FUNCTION_BLOCK NeredaSludgeBuffer (* Composite Function Block Type *)
  (* Standard: 61499-2 *)
  (* Version 0.0, 4/25/2024, SESA713705, Schneider Electric, template *)
  PACKAGE SE.Nereda;
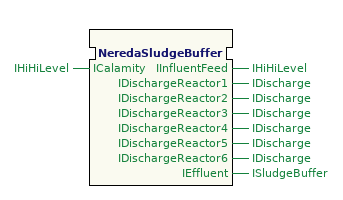
  SOCKETS
    ICalamity : IHiHiLevel;
  END_SOCKETS
  PLUGS
    IInfluentFeed : IHiHiLevel;
    IDischargeReactor1 : IDischarge;
    IDischargeReactor2 : IDischarge;
    IDischargeReactor3 : IDischarge;
    IDischargeReactor4 : IDischarge;
    IDischargeReactor5 : IDischarge;
    IDischargeReactor6 : IDischarge;
    IEffluent : ISludgeBuffer; (* Process value and status interface adapter *)
  END_PLUGS
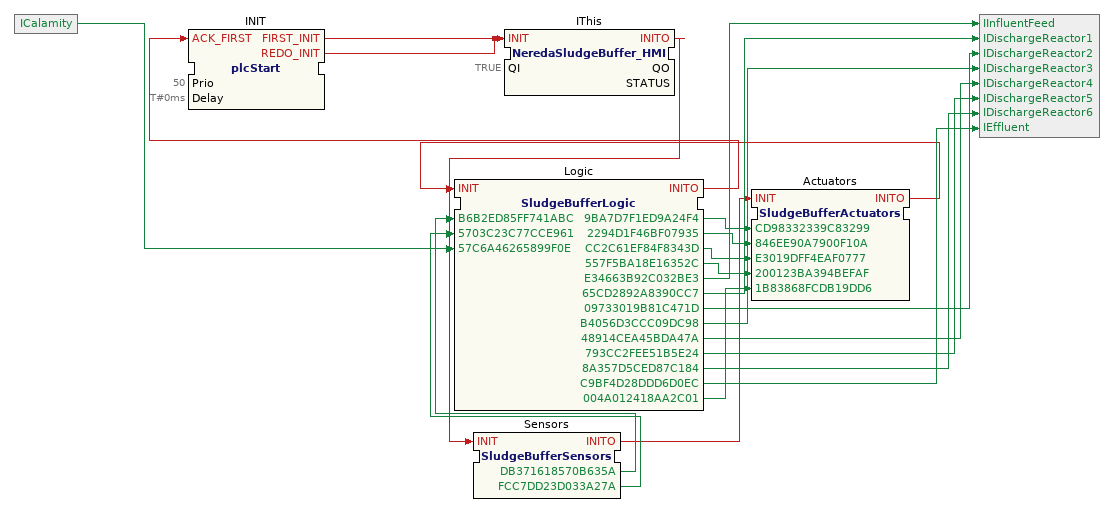
  (* 01 - FUNCTIONNAL INPUT INTERFACE *)
  (* 00 - INITIALIZATION *)
  (* 05 - LOGIC *)
  (* 06 - HMI INTERFACE *)
  (* 03 - FIELD INTERFACE *)
  (* 02 - FUNCTIONNAL OUTPUT INTERFACE *)
  (* Sludge Buffer Logic *)
  (* 04 - CHILDREN *)
  (* 4A - TYPICALS *)
  FBS
    IThis : NeredaSludgeBuffer_HMI(QI := TRUE);
    INIT : plcStart(Prio := 50, Delay := T#0ms);
    Actuators : SludgeBufferActuators;
    Sensors : SludgeBufferSensors;
    Logic : SludgeBufferLogic;
  END_FBS
  EVENT_CONNECTIONS
    INIT.FIRST_INIT TO IThis.INIT;
    INIT.REDO_INIT TO IThis.INIT;
    IThis.INITO TO Sensors.INIT;
    Actuators.INITO TO Logic.INIT;
    Logic.INITO TO INIT.ACK_FIRST;
    Sensors.INITO TO Actuators.INIT;
  END_CONNECTIONS
  ADAPTER_CONNECTIONS
    Sensors.DB371618570B635A TO Logic.B6B2ED85FF741ABC;
    Sensors.FCC7DD23D033A27A TO Logic.5703C23C77CCE961;
    ICalamity TO Logic.57C6A46265899F0E;
    Logic.9BA7D7F1ED9A24F4 TO Actuators.CD98332339C83299;
    Logic.2294D1F46BF07935 TO Actuators.846EE90A7900F10A;
    Logic.CC2C61EF84F8343D TO Actuators.E3019DFF4EAF0777;
    Logic.557F5BA18E16352C TO Actuators.200123BA394BEFAF;
    Logic.E34663B92C032BE3 TO IInfluentFeed;
    Logic.65CD2892A8390CC7 TO IDischargeReactor1;
    Logic.09733019B81C471D TO IDischargeReactor2;
    Logic.B4056D3CCC09DC98 TO IDischargeReactor3;
    Logic.48914CEA45BDA47A TO IDischargeReactor4;
    Logic.793CC2FEE51B5E24 TO IDischargeReactor5;
    Logic.8A357D5CED87C184 TO IDischargeReactor6;
    Logic.C9BF4D28DDD6D0EC TO IEffluent;
    Logic.004A012418AA2C01 TO Actuators.1B83868FCDB19DD6;
  END_CONNECTIONS
END_FUNCTION_BLOCK
